// Mitsubishi GX Works2 project: z06   PLC: Q02/Q02H

PROGRAM MAIN
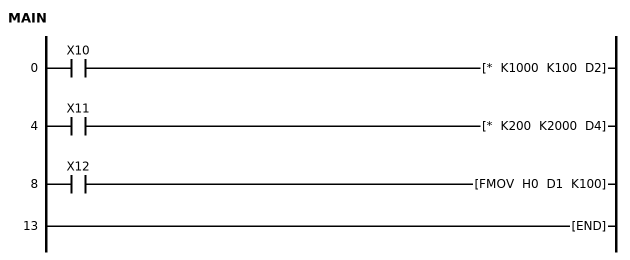
0     LD      X10
      *       K1000 K100 D2
4     LD      X11
      *       K200 K2000 D4
8     LD      X12
      FMOV    H0 D1 K100
13    END
END_PROGRAM
